INTERFACE PUBLIC I_JogMoveBuilder EXTENDS __System.IQueryInterface

METHOD PUBLIC Acceleration : I_MoveBuilder
VAR_INPUT
	value : LREAL;
END_VAR
END_METHOD

METHOD PUBLIC BuildBackwardsCommand : I_MoveCommand
END_METHOD

METHOD PUBLIC BuildForwardCommand : I_MoveCommand
END_METHOD

METHOD PUBLIC Deceleration : I_MoveBuilder
VAR_INPUT
	value : LREAL;
END_VAR
END_METHOD

METHOD PUBLIC Distance : I_JogMoveBuilder
VAR_INPUT
	value : LREAL;
END_VAR
END_METHOD

METHOD PUBLIC Jerk : I_MoveBuilder
VAR_INPUT
	value : LREAL;
END_VAR
END_METHOD

METHOD PUBLIC Velocity : I_MoveBuilder
VAR_INPUT
	value : LREAL;
END_VAR
END_METHOD

END_INTERFACE

(* stored: Version 1.1.0.1, ProductVersion 3.1.4024.12
   Itf I_JogMoveBuilder: Id {74434c50-6753-4844-97d0-c27a98431a9c}
   Method Acceleration: Id {d649dbf4-d723-4c50-912a-2f5aed25b170}
   Method BuildBackwardsCommand: Id {aafd07e9-f6b3-4356-8088-e1f73610b6cf}
   Method BuildForwardCommand: Id {58a3b487-076f-48e0-8cb8-8b8988e38fe7}
   Method Deceleration: Id {59da1220-7ac2-4382-8265-df82076960d0}
   Method Distance: Id {6de70f7f-321d-4d45-840b-73778016af0a}
   Method Jerk: Id {bcdecc2d-b389-44ae-82c3-f03458ffddbf}
   Method Velocity: Id {90689bf3-1272-471d-80e5-ba1393d6e9d7} *)
